(* CODESYS project SLL_IFM_Version_SP11p0.library
   Author: adam@sperrinlogic.com
   Version: 0.0.0.2
   Title: SLL_IFM_Version
   DefaultNamespace: SLL_IFM_Version
   Placeholder: SLL_IFM_Version
   Company: SLL

Project tree, tasks and I/O mapping:
  libraries: Util, 3.5.19.0 (System); Standard, 3.5.18.0 (System); ifmTypes, 1.9.6.0 (ifm electronic); CmpApp, 3.5.17.0 (System); ifmRawCAN, 4.0.3.0 (ifm electronic); ifmDeviceCR07nn, 1.2.2.0 (ifm electronic); SysTarget, 3.5.17.0 (System); SysTypes2 Interfaces, * (System)
  STRUCTS/
    data type PLC_Version
  FUNCS/
    program Get_Version_Struct [ST]
    program PLC_System_Info [ST]
    function block PLC_Version_Unpack_FB [ST]
*)

// STRUCTS/PLC_Version
TYPE PLC_Version :
STRUCT
	IsReleased: BOOL;	
	Machine: STRING(20);
	Hardware: STRING(20);
	Info: STRING(20);
    verCompiler : VERSION;
    verRuntime : VERSION;
	ProjectName : STRING;
	Author : STRING;
	Version : STRING;
	Description : STRING;
	Profile : STRING;
	LastChanges :STRING;
END_STRUCT
END_TYPE

// FUNCS/Get_Version_Struct
PROGRAM Get_Version_Struct
VAR
	AppIECResult: CmpApp.RTS_IEC_RESULT;
	AppInfoIECResult: CmpApp.RTS_IEC_RESULT;
	AppPtr: POINTER TO APPLICATION_INFO;
END_VAR
VAR_INPUT
	pMachine: STRING(20);
	pHardware: STRING(20);
	pInfo: STRING(20);
	pIsReleased: BOOL;
	pCompileDateTime: WSTRING;
END_VAR
VAR_OUTPUT
	pStruct: PLC_Version;
END_VAR

pStruct.verRuntime := __SYSTEM.Constants.RuntimeVersion;
pStruct.verCompiler := __SYSTEM.Constants.CompilerVersion;
AppPtr := CmpApp.AppGetApplicationInfo(CmpApp.AppGetCurrent(ADR(AppIECResult)),ADR(AppInfoIECResult));

IF AppInfoIECResult = 0 THEN
	pStruct.ProjectName:=AppPtr^.pstProjectName^;				
	pStruct.Author:=AppPtr^.pstAuthor^;
	pStruct.Version:=AppPtr^.pstVersion^;
	pStruct.Description:=AppPtr^.pstDescription^;
	pStruct.Profile:=AppPtr^.pstProfile^;
END_IF

pStruct.LastChanges:=TO_STRING(pCompileDateTime);
pStruct.IsReleased := pIsReleased;
pStruct.Machine:=pMachine;
pStruct.Hardware:=pHardware;
pStruct.Info:=pInfo;

END_PROGRAM

// FUNCS/PLC_System_Info
PROGRAM PLC_System_Info
VAR
    dwType          : DWORD;
    dwId            : DWORD;
    dwVersion       : DWORD;
    iecResult       : UDINT;
 
    wName           : WSTRING;
    udiNameLength   : UDINT := 80;
 
    udiOsInfo       : UDINT := 80;
	NameLen:INT;
END_VAR

VAR_OUTPUT
	PC_SIM: INT;
END_VAR


iecResult := SysTargetGetType(ADR(dwType));
iecResult := SysTargetGetId(ADR(dwId));
 
iecResult := SysTargetGetVendorName(ADR(wName),ADR(udiNameLength));
iecResult := SysTargetGetVersion(ADR(dwVersion));
 
udiOsInfo := SysTargetGetOperatingSystemId(ADR(udiOsInfo));

NameLen := LEN(WSTRING_TO_STRING(wName));

IF NameLen = 0 THEN
	PC_SIM:=1;
ELSE
	PC_SIM:=0;	
END_IF

END_PROGRAM

// FUNCS/PLC_Version_Unpack_FB
FUNCTION_BLOCK PLC_Version_Unpack_FB
VAR_INPUT
	pVersion: REFERENCE TO PLC_Version;
END_VAR
VAR_OUTPUT
	oMachine:STRING;
	oCompiler:STRING;
	oVersion:STRING;
END_VAR
VAR
	tempCompiler:STRING;
	tempRuntime:STRING;
END_VAR

oMachine:='';
oMachine:=CONCAT(oMachine,pVersion.ProjectName);
oMachine:=CONCAT(oMachine,',');
oMachine:=CONCAT(oMachine,pVersion.Machine);
oMachine:=CONCAT(oMachine,',');
oMachine:=CONCAT(oMachine,pVersion.Hardware);
oMachine:=CONCAT(oMachine,',');
oMachine:=CONCAT(oMachine,pVersion.Info);

oVersion:='Version:';
oVersion:=CONCAT(oVersion,pVersion.Version);
oVersion:=CONCAT(oVersion,',(');
oVersion:=CONCAT(oVersion,pVersion.LastChanges);
oVersion:=CONCAT(oVersion,'),');
IF pVersion.IsReleased THEN
	oVersion:=CONCAT(oVersion,'Release');
ELSE
	oVersion:=CONCAT(oVersion,'Debug');	
END_IF

tempRuntime:='';
tempRuntime:=CONCAT(tempRuntime,TO_STRING(pVersion.verRuntime.uiMajor));
tempRuntime:=CONCAT(tempRuntime,'.');
tempRuntime:=CONCAT(tempRuntime,TO_STRING(pVersion.verRuntime.uiMinor));
tempRuntime:=CONCAT(tempRuntime,'.');
tempRuntime:=CONCAT(tempRuntime,TO_STRING(pVersion.verRuntime.uiPatch));
tempRuntime:=CONCAT(tempRuntime,'.');
tempRuntime:=CONCAT(tempRuntime,TO_STRING(pVersion.verRuntime.uiServicePack));

tempCompiler:='';
tempCompiler:=CONCAT(tempCompiler,TO_STRING(pVersion.verCompiler.uiMajor));
tempCompiler:=CONCAT(tempCompiler,'.');
tempCompiler:=CONCAT(tempCompiler,TO_STRING(pVersion.verCompiler.uiMinor));
tempCompiler:=CONCAT(tempCompiler,'.');
tempCompiler:=CONCAT(tempCompiler,TO_STRING(pVersion.verCompiler.uiPatch));
tempCompiler:=CONCAT(tempCompiler,'.');
tempCompiler:=CONCAT(tempCompiler,TO_STRING(pVersion.verCompiler.uiServicePack));

oCompiler:='Compiler:';
oCompiler:=CONCAT(oCompiler,tempCompiler);
oCompiler:=CONCAT(oCompiler,',Runtime:');
oCompiler:=CONCAT(oCompiler,tempRuntime);

END_FUNCTION_BLOCK
